FUNCTION_BLOCK Room_State_Idle EXTENDS Room_State
VAR_INPUT
END_VAR
VAR_OUTPUT
END_VAR
VAR
END_VAR

METHOD OnInit
_ctx.io.out.bInletValve := FALSE;
_ctx.io.out.bOutletValve := FALSE;

_ctx.priv.bAbort := TRUE;
END_METHOD

END_FUNCTION_BLOCK

(* stored: Version 1.1.0.1
   POU Room_State_Idle: Id {4c766015-91cf-477b-985f-581e4af963c5}, SpecialFunc None
   Method OnInit: Id {d4b48581-1a4d-4829-a23f-cfc37a8808cd} *)
